SUBAPPLICATION I_GetAttribute_IDA (* Bündelung von I_GetAttribute (Kommando GetAttribute F.58) und Attribute_IDA (asynchroner Adapter-Empfang) mit gemeinsamen u16ObjId und u8AID Parametern *)
  (* Standard: 61499-2; Description: Copyright (c) 2026 Meisterschulen am Ostbahnhof This program and the accompanying materials are made available under the terms of the Eclipse Public License 2.0 which is available at https://www.eclipse.org/legal/epl-2.0/ SPDX-License-Identifier: EPL-2.0 *)
  (* Version 1.0, 2026-09-15, Franz Höpfinger, Meisterschulen am Ostbahnhof, Initial implementation combining I_GetAttribute and Attribute_IDA *)
  PACKAGE MyLib::sys;
  IMPORT isobus::UT::Q::const::IDs::ID_NULL;
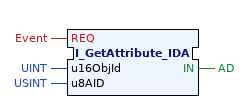
  EVENT_INPUT
    REQ; (* Service Request *)
  END_EVENT
  VAR_INPUT
    u16ObjId : UINT := ID_NULL; (* Object ID *)
    u8AID : USINT; (* Attribute ID of the object *)
  END_VAR
  PLUGS
    IN : adapter::types::unidirectional::AD; (* Input data from resource *)
  END_PLUGS
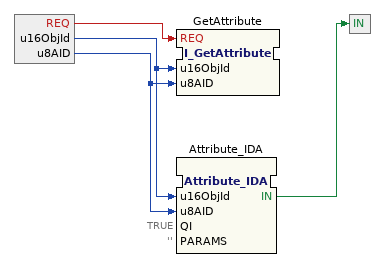
  FBS
    GetAttribute : isobus::UT::I::I_GetAttribute;
    Attribute_IDA : isobus::UT::io::Attribute::Attribute_IDA(QI := TRUE, PARAMS := '');
  END_FBS
  EVENT_CONNECTIONS
    REQ TO GetAttribute.REQ;
  END_CONNECTIONS
  DATA_CONNECTIONS
    u16ObjId TO GetAttribute.u16ObjId;
    u16ObjId TO Attribute_IDA.u16ObjId;
    u8AID TO GetAttribute.u8AID;
    u8AID TO Attribute_IDA.u8AID;
  END_CONNECTIONS
  ADAPTER_CONNECTIONS
    Attribute_IDA.IN TO IN;
  END_CONNECTIONS
END_SUBAPPLICATION
